Fanuc KAREL source: kt00020.KL

-- PROVISIONAL review KL for V940-1; original PC SHA256 cc8e9fbb1988943448d2da6330cffaaa4b81ab43c7bf91b68e97cf19bb3db706
-- Incomplete behavior may be omitted. Consult companion uncertainty JSON. Do not deploy.
PROGRAM KT00020
%NOLOCKGROUP
VAR
  R2 : REAL
  OUT : REAL
-- UNRESOLVED_DECL Y1 type=002018
BEGIN
  -- V9_ZERO_TABLE_METADATA_HINT layout=0001; no indexed target words; source/name/runtime held
  -- UNRESOLVED_PC offsets 5-19; opcodes 2E,22,9D,33,B2
  -- UNRESOLVED_PC offsets 24-35; opcodes 2E,23
  -- UNRESOLVED_PC offsets 40-64; opcodes 22,9D,33,B1,21,29,64,69,23
  -- UNRESOLVED_PC offsets 69-73; opcodes 7F
END KT00020
